# EPICS substitutions: fastFeedbackApp/Db/common/fbckSettledSum.substitutions
file fbckSettledStatus.template {
        pattern { LOOP }
                { $(LP)}
}
